INTERFACE I_Dome

PROPERTY Capabilities : INT
GET
END_GET
END_PROPERTY

METHOD Close : BOOL
VAR_INPUT
END_VAR
END_METHOD

PROPERTY Error : BOOL
GET
END_GET
END_PROPERTY

PROPERTY ErrorID : UDINT
GET
END_GET
END_PROPERTY

METHOD Open : BOOL
VAR_INPUT
END_VAR
END_METHOD

METHOD Park : BOOL
VAR_INPUT
END_VAR
END_METHOD

PROPERTY Parked : BOOL
GET
END_GET
END_PROPERTY

PROPERTY Position : LREAL
GET
END_GET
SET
END_SET
END_PROPERTY

METHOD Reset : BOOL
VAR_INPUT
END_VAR
END_METHOD

PROPERTY RotState : E_DomeRotationState
GET
END_GET
END_PROPERTY

PROPERTY ShutterState : E_RoofState
GET
END_GET
SET
END_SET
END_PROPERTY

METHOD Stop : BOOL
VAR_INPUT
END_VAR
END_METHOD

METHOD StopTrack : BOOL
VAR_INPUT
END_VAR
END_METHOD

METHOD Track : BOOL
VAR_INPUT
END_VAR
END_METHOD

PROPERTY Tracking : BOOL
GET
END_GET
END_PROPERTY

END_INTERFACE

(* stored: Version 1.1.0.1, ProductVersion 3.1.4024.15
   Itf I_Dome: Id {97c41eeb-cc9f-4286-aebb-137faba3b329}
   Property Capabilities: Id {ce62be83-41b1-484e-96cb-80c465df6602}
   Get Get: Id {4f2a8459-f8db-47dc-a316-699a4621e3d7}
   Method Close: Id {324da6d9-cec6-4890-ad47-67782826b0a8}
   Property Error: Id {a794a4bc-62d7-45f0-94ee-2879b59d67e9}
   Get Get: Id {d77664c7-c8dc-4360-a991-27233099243e}
   Property ErrorID: Id {23f972b2-0650-45e6-9f00-215590f68f85}
   Get Get: Id {dc7d32e9-a08e-4407-b52b-6af80e99487b}
   Method Open: Id {93be79ba-c7cb-4bb7-a779-5569a9b5f64b}
   Method Park: Id {ec477463-5cda-448f-946a-095caeb42b46}
   Property Parked: Id {b36a6845-c8da-493a-807b-13e34dcb1c3c}
   Get Get: Id {3d26b278-b164-42c8-ac02-0f45a894de74}
   Property Position: Id {fcad9bb1-0998-4626-b0b3-b366fd66317a}
   Get Get: Id {2bb94df7-ad12-49df-852c-47e0779ed164}
   Set Set: Id {2a48082d-c172-4984-bad0-748564b2bd51}
   Method Reset: Id {7cb5034b-2625-4d18-b1cd-4cf4aad842da}
   Property RotState: Id {7210269f-3287-4ee9-b4b6-ea62cb9473cb}
   Get Get: Id {bc306067-186a-4fbf-a0b9-cf743eb5905f}
   Property ShutterState: Id {06ad0786-c570-473f-8ca9-4a5d10920604}
   Get Get: Id {2925be68-4591-4226-8720-0f7cd5ff2baf}
   Set Set: Id {12de55ee-1a05-45b5-ba14-f4fd6b06663b}
   Method Stop: Id {606de154-cb59-41c6-bfba-af948b1ef0cc}
   Method StopTrack: Id {db4faf08-b158-4f1f-882a-1c0ed13959f6}
   Method Track: Id {bf111ab9-334e-415e-b99d-0bdc6457753a}
   Property Tracking: Id {3c48ab71-271d-4230-8284-85891e3c766d}
   Get Get: Id {aa429e62-32dc-4010-a0a4-4357cce9602e} *)
